// TIA Portal V15.1 export
// export: Created 2024-05-17T05:38:52.6374958Z, ExportSetting WithDefaults, DisplayName Totally Integrated Automation Portal, DisplayVersion V15.1 Update 5, DisplayName TIA Portal Openness, DisplayVersion V15.1 Update 5, DisplayName SINAMICS Startdrive Advanced, DisplayVersion V15.1, DisplayName G130, G150, S120, S150, SINAMICS MV, S210, DisplayVersion V15.1, DisplayName G110M, G120, G120C, G120D, G120P, DisplayVersion V15.1, DisplayName STEP 7 Professional, DisplayVersion V15.1 Update 5, DisplayName STEP 7 Safety, DisplayVersion V15.1, DisplayName WinCC Professional, DisplayVersion V15.1 Update 5, DisplayName SIMATIC Visualization Architect, DisplayVersion V15.1
FUNCTION_BLOCK "LGBTrfOutRel"   // FB6701, FBD
TITLE = LGBTrfOutRel
{ S7_Optimized_Access := 'TRUE' }
VERSION : 0.1
// =============================================================================
// The ReleaseTrfOut function is a FB to be used in transport functions 
// block (as roller, cross-section, …) to release an OUT transfer at an earlier
// stage to gain cycletime in automatic Mode or in manual Mode.
// stored: AutoNumber false, IsIECCheckEnabled false, IsRetainMemResEnabled false, MemoryReserve 100, SetENOAutomatically False, UDAEnableTagReadback false
   VAR_INPUT
      I_TrfOutPrev_TM { ExternalAccessible := 'False'; ExternalVisible := 'False'; ExternalWritable := 'False'} : Bool;   // Transfer communication for outfeed from previous conveyor
      I_TrfOutPrev_RdyDlv { ExternalAccessible := 'False'; ExternalVisible := 'False'; ExternalWritable := 'False'} : Bool;   // Transfer communication for outfeed from previous conveyor
      I_TrfInNext_Arrived { ExternalAccessible := 'False'; ExternalVisible := 'False'; ExternalWritable := 'False'} : Bool;   // Transfer communication for infeed on next conveyor
      I_TrfInNext_RdyRcv { ExternalAccessible := 'False'; ExternalVisible := 'False'; ExternalWritable := 'False'} : Bool;   // Transfer communication for infeed on next conveyor
      I_ReleaseDet { ExternalAccessible := 'False'; ExternalVisible := 'False'; ExternalWritable := 'False'} : Bool;   // Detection to release the outfeed transfer of the previous conveyor
      I_SafetyOk { ExternalAccessible := 'False'; ExternalVisible := 'False'; ExternalWritable := 'False'} : Bool;   // Safety Ok
   END_VAR
   VAR_OUTPUT
      O_TrfOutPrev_Arrived { ExternalAccessible := 'False'; ExternalVisible := 'False'; ExternalWritable := 'False'} : Bool;   // Transfer communication for outfeed from previous conveyor
      O_TrfOutPrev_RdyRcv { ExternalAccessible := 'False'; ExternalVisible := 'False'; ExternalWritable := 'False'} : Bool;   // Transfer communication for outfeed from previous conveyor
      O_TrfInNext_TrfOutCmd { ExternalAccessible := 'False'; ExternalVisible := 'False'; ExternalWritable := 'False'} : Bool;   // Command request after interlock / Command Request after Interlock / Transfer communication for infeed on next conveyor
      O_TrfInNext_TM { ExternalAccessible := 'False'; ExternalVisible := 'False'; ExternalWritable := 'False'} : Bool;   // Transfer communication for infeed on next conveyor
      O_TrfInNext_RdyDlv { ExternalAccessible := 'False'; ExternalVisible := 'False'; ExternalWritable := 'False'} : Bool;   // Transfer communication for infeed on next conveyor
      O_OvertimeAlarm { ExternalAccessible := 'False'; ExternalVisible := 'False'; ExternalWritable := 'False'} : Bool;   // Overtime alarm (0=no alarm / 1=Alarm) / Overtime Alarm
      O_ConfigCalibrationAlm { ExternalAccessible := 'False'; ExternalVisible := 'False'; ExternalWritable := 'False'} : Bool;   // Config/Calibration Alarm
      O_CalibrationWarn { ExternalAccessible := 'False'; ExternalVisible := 'False'; ExternalWritable := 'False'} : Bool;   // Warning Calibration
      O_AlarmABCondition { ExternalAccessible := 'False'; ExternalVisible := 'False'; ExternalWritable := 'False'} : Bool;   // Alarm AB condition / Alarm AB Condition
   END_VAR
   VAR_IN_OUT
      IO_Modes : "Modes";   // Modes
      H_HMI : "H_HMI";   // Animation
      H_TrfOut : "H_TrfOut";   // Animation
      C_TrfMaxTime { ExternalAccessible := 'False'; ExternalVisible := 'False'; ExternalWritable := 'False'} : DInt := 8000;   // Time Delay-On Overtime alarm (millisec) / Time Delay-On Overtime Alarm (millisec)
      C_TrfMaxTimeAfterOvertime { ExternalAccessible := 'False'; ExternalVisible := 'False'; ExternalWritable := 'False'} : DInt := 0;   // Time Delay-On after reset/start after Overtime Alarm (millisec)
      C_EnableTimeoutAlarm { ExternalAccessible := 'False'; ExternalVisible := 'False'; ExternalWritable := 'False'} : Bool;   // Enable Timeout Alarm
   END_VAR
   VAR RETAIN
      Release { ExternalAccessible := 'False'; ExternalVisible := 'False'; ExternalWritable := 'False'} : Bool;   // Memory of release detection negative edge
   END_VAR
   VAR
      Edge { ExternalAccessible := 'False'; ExternalVisible := 'False'; ExternalWritable := 'False'} : Array[0..3] of Bool;   // Edges
      AlarmA { ExternalAccessible := 'False'; ExternalVisible := 'False'; ExternalWritable := 'False'} : Bool;   // Summation Alarm A of roller. / Alarm A
      AlarmB { ExternalAccessible := 'False'; ExternalVisible := 'False'; ExternalWritable := 'False'} : Bool;   // Summation Alarm B of roller. / Alarm B
      AlarmC { ExternalAccessible := 'False'; ExternalVisible := 'False'; ExternalWritable := 'False'} : Bool;   // Summation Alarm C of roller. / Alarm C
      AlarmD { ExternalAccessible := 'False'; ExternalVisible := 'False'; ExternalWritable := 'False'} : Bool;   // Summation Alarm D of roller. / Alarm D
      AlarmABCondition { ExternalAccessible := 'False'; ExternalVisible := 'False'; ExternalWritable := 'False'} : Bool;   // Resetable alarm / Alarm AB Condition
   END_VAR
   VAR RETAIN
      OvertimeAlarm { ExternalAccessible := 'False'; ExternalVisible := 'False'; ExternalWritable := 'False'} : Bool;   // MEM Overtime alarm / MEM Overtime Alarm
      OvertimeAlarmAlmCond { ExternalAccessible := 'False'; ExternalVisible := 'False'; ExternalWritable := 'False'} : Bool;   // MEM Overtime alarm / MEM Overtime Alarm / Overtime Alarm
      TimerOvertimeAlarm { ExternalAccessible := 'False'; ExternalVisible := 'False'; ExternalWritable := 'False'} : Bool;   // MEM Overtime alarm / MEM Overtime Alarm / Overtime Alarm
   END_VAR
   VAR
      TimerOvertimAlarm { ExternalAccessible := 'False'; ExternalVisible := 'False'; ExternalWritable := 'False'} : "LTimer";   // FB
      TrfMaxTime { ExternalAccessible := 'False'; ExternalVisible := 'False'; ExternalWritable := 'False'} : DInt;   // Maximum Transfer Time
      ConfigCalibrationAlm { ExternalAccessible := 'False'; ExternalVisible := 'False'; ExternalWritable := 'False'} : Bool;   // Config/Calibration Alarm
      CalibrationWarn { ExternalAccessible := 'False'; ExternalVisible := 'False'; ExternalWritable := 'False'} : Bool;   // Warning Calibration
   END_VAR
   VAR RETAIN
      OvtTrfMaxTime { ExternalAccessible := 'False'; ExternalVisible := 'False'; ExternalWritable := 'False'} : DInt;   // Alarm Value
      OvtTrfMaxTimeAfterOvertime { ExternalAccessible := 'False'; ExternalVisible := 'False'; ExternalWritable := 'False'} : DInt;   // Alarm Value
      CalibratedTransfer { ExternalAccessible := 'False'; ExternalVisible := 'False'; ExternalWritable := 'False'} : Bool;
   END_VAR
   VAR
      AlarmTimeWithConfig { ExternalAccessible := 'False'; ExternalVisible := 'False'; ExternalWritable := 'False'} : Bool;
      AlarmTimeWithCalibration { ExternalAccessible := 'False'; ExternalVisible := 'False'; ExternalWritable := 'False'} : Bool;
   END_VAR
   VAR_TEMP
      H_CalibrateTransfer : Bool;   // HMI Function
      TempReal : Real;
   END_VAR
   VAR_TEMP   // added for the SCL form of the ladder/FBD networks
      _w1 : Bool;
      _w2 : Bool;
      _w3 : Bool;
      _w4 : Bool;
   END_VAR
BEGIN

REGION Network 1: **** 1 - Inputs **** HMI Commands
   // Extract the Commands from HMIRobCmd / Extract the Commands from HMI
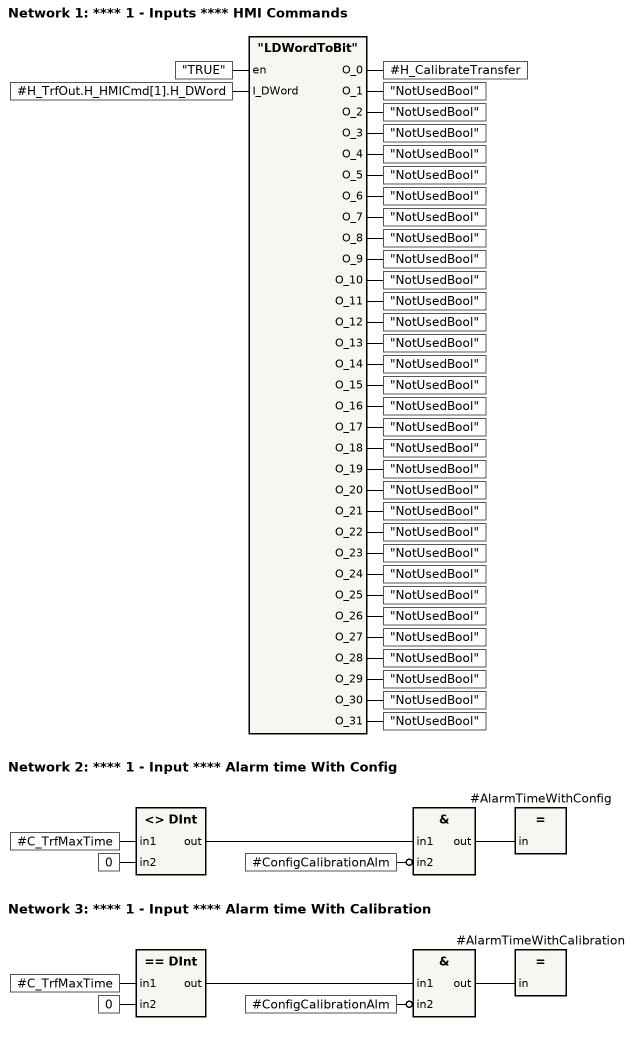
   IF "TRUE" THEN
       "LDWordToBit"(I_DWord := #H_TrfOut.H_HMICmd[1].H_DWord,
                     O_0 => #H_CalibrateTransfer,
                     O_1 => "NotUsedBool",
                     O_2 => "NotUsedBool",
                     O_3 => "NotUsedBool",
                     O_4 => "NotUsedBool",
                     O_5 => "NotUsedBool",
                     O_6 => "NotUsedBool",
                     O_7 => "NotUsedBool",
                     O_8 => "NotUsedBool",
                     O_9 => "NotUsedBool",
                     O_10 => "NotUsedBool",
                     O_11 => "NotUsedBool",
                     O_12 => "NotUsedBool",
                     O_13 => "NotUsedBool",
                     O_14 => "NotUsedBool",
                     O_15 => "NotUsedBool",
                     O_16 => "NotUsedBool",
                     O_17 => "NotUsedBool",
                     O_18 => "NotUsedBool",
                     O_19 => "NotUsedBool",
                     O_20 => "NotUsedBool",
                     O_21 => "NotUsedBool",
                     O_22 => "NotUsedBool",
                     O_23 => "NotUsedBool",
                     O_24 => "NotUsedBool",
                     O_25 => "NotUsedBool",
                     O_26 => "NotUsedBool",
                     O_27 => "NotUsedBool",
                     O_28 => "NotUsedBool",
                     O_29 => "NotUsedBool",
                     O_30 => "NotUsedBool",
                     O_31 => "NotUsedBool");
   END_IF;
END_REGION

REGION Network 2: **** 1 - Input **** Alarm time With Config
   #AlarmTimeWithConfig := (#C_TrfMaxTime <> 0) AND NOT #ConfigCalibrationAlm;
END_REGION

REGION Network 3: **** 1 - Input **** Alarm time With Calibration
   #AlarmTimeWithCalibration := (#C_TrfMaxTime = 0) AND NOT #ConfigCalibrationAlm;
END_REGION

REGION Network 4: Calibrated Set / **** 1 - Input **** Ovt Values / **** 1 - Inputs **** Ovt Values
   // Ovt Values
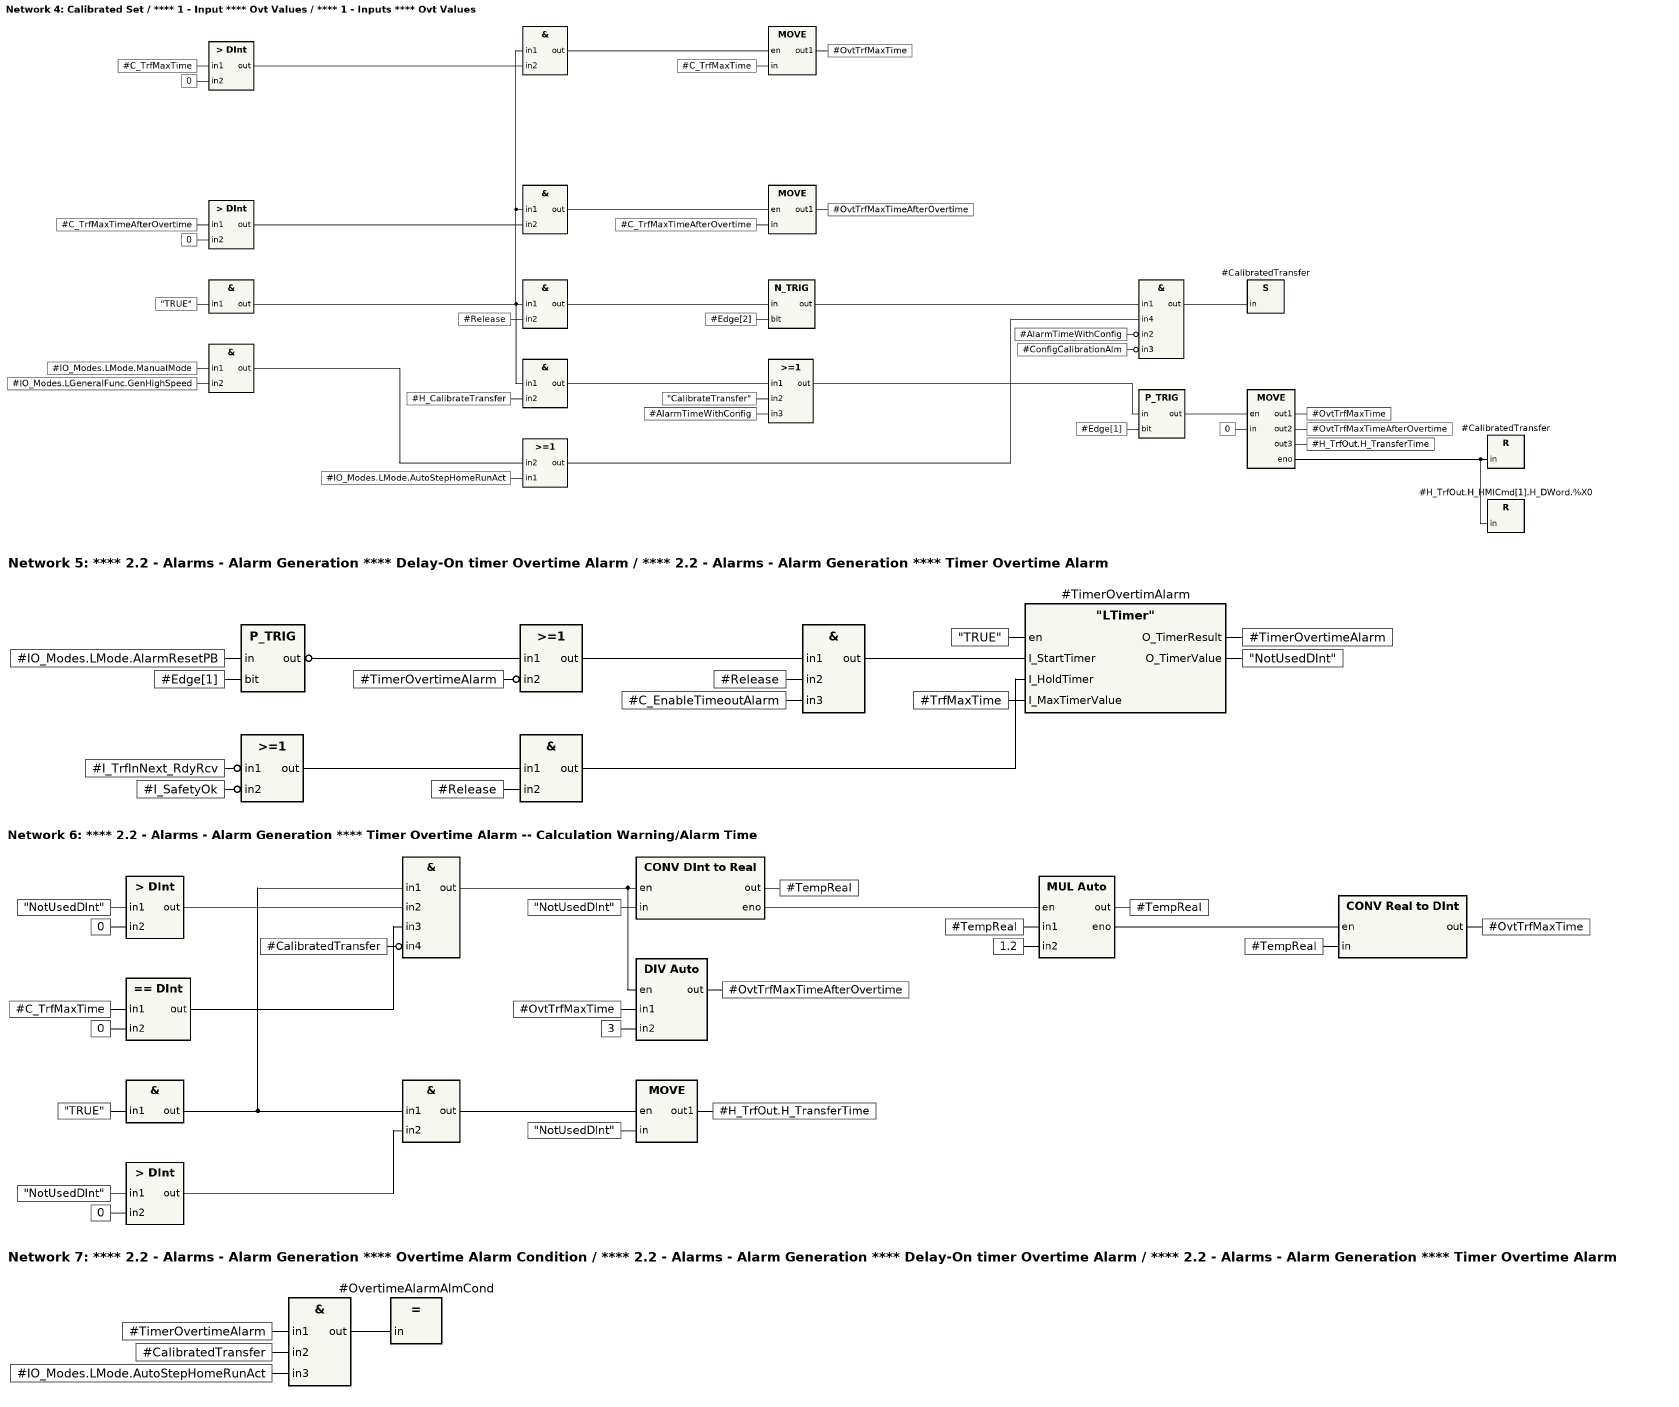
   // ENO of a box is taken as its EN; it also drops when the box reports an error
   IF "TRUE" AND (#C_TrfMaxTime > 0) THEN #OvtTrfMaxTime := #C_TrfMaxTime; END_IF;
   IF "TRUE" AND (#C_TrfMaxTimeAfterOvertime > 0) THEN
       #OvtTrfMaxTimeAfterOvertime := #C_TrfMaxTimeAfterOvertime;
   END_IF;
   #_w1 := "TRUE" AND #Release;
   #_w2 := NOT #_w1 AND #Edge[2];   // falling edge
   #Edge[2] := #_w1;
   IF #_w2 AND ((#IO_Modes.LMode.ManualMode AND #IO_Modes.LGeneralFunc.GenHighSpeed) OR #IO_Modes.LMode.AutoStepHomeRunAct) AND NOT #AlarmTimeWithConfig AND NOT #ConfigCalibrationAlm THEN
       #CalibratedTransfer := TRUE;
   END_IF;
   #_w3 := ("TRUE" AND #H_CalibrateTransfer) OR "CalibrateTransfer" OR #AlarmTimeWithConfig;
   #_w4 := #_w3 AND NOT #Edge[1];   // rising edge
   #Edge[1] := #_w3;
   IF #_w4 THEN
       #OvtTrfMaxTime := 0;
       #OvtTrfMaxTimeAfterOvertime := 0;
       #H_TrfOut.H_TransferTime := 0;
       #CalibratedTransfer := FALSE;
       #H_TrfOut.H_HMICmd[1].H_DWord.%X0 := FALSE;
   END_IF;
END_REGION

REGION Network 5: **** 2.2 - Alarms - Alarm Generation **** Delay-On timer Overtime Alarm / **** 2.2 - Alarms - Alarm Generation **** Timer Overtime Alarm
   // Delay-On timer Overtime Alarm
   #_w1 := #IO_Modes.LMode.AlarmResetPB AND NOT #Edge[1];   // rising edge
   #Edge[1] := #IO_Modes.LMode.AlarmResetPB;
   IF "TRUE" THEN
       #TimerOvertimAlarm(I_StartTimer := (NOT #_w1 OR NOT #TimerOvertimeAlarm) AND #Release AND #C_EnableTimeoutAlarm,   // "LTimer"
                          I_HoldTimer := (NOT #I_TrfInNext_RdyRcv OR NOT #I_SafetyOk) AND #Release,
                          I_MaxTimerValue := #TrfMaxTime,
                          O_TimerResult => #TimerOvertimeAlarm,
                          O_TimerValue => "NotUsedDInt");
   END_IF;
END_REGION

REGION Network 6: **** 2.2 - Alarms - Alarm Generation **** Timer Overtime Alarm -- Calculation Warning/Alarm Time
   IF "TRUE" AND ("NotUsedDInt" > 0) AND (#C_TrfMaxTime = 0) AND NOT #CalibratedTransfer THEN
       #TempReal := DINT_TO_REAL("NotUsedDInt");
       #TempReal := #TempReal * 1.2;
       #OvtTrfMaxTime := REAL_TO_DINT(#TempReal);
       #OvtTrfMaxTimeAfterOvertime := #OvtTrfMaxTime / 3;
   END_IF;
   IF "TRUE" AND ("NotUsedDInt" > 0) THEN #H_TrfOut.H_TransferTime := "NotUsedDInt"; END_IF;
END_REGION

REGION Network 7: **** 2.2 - Alarms - Alarm Generation **** Overtime Alarm Condition / **** 2.2 - Alarms - Alarm Generation **** Delay-On timer Overtime Alarm / **** 2.2 - Alarms - Alarm Generation **** Timer Overtime Alarm
   // Delay-On timer Overtime Alarm
   #OvertimeAlarmAlmCond := #TimerOvertimeAlarm AND #CalibratedTransfer AND #IO_Modes.LMode.AutoStepHomeRunAct;
END_REGION

REGION Network 8: **** 2.2 - Alarms - Alarm Generation **** OverTime Alarm / **** 2.2 - Alarms - Alarm Generation **** Overrtime Alarm
   // Overrtime Alarm
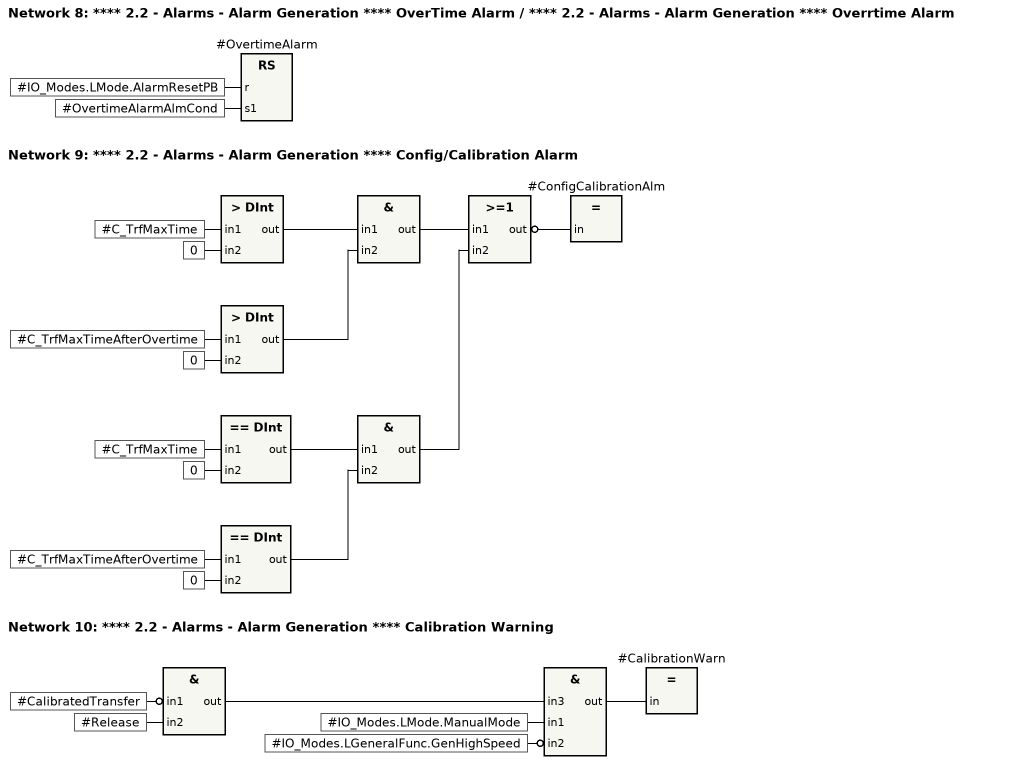
   IF #IO_Modes.LMode.AlarmResetPB THEN
       #OvertimeAlarm := FALSE;   // RS flip-flop
   END_IF;
   IF #OvertimeAlarmAlmCond THEN #OvertimeAlarm := TRUE; END_IF;
END_REGION

REGION Network 9: **** 2.2 - Alarms - Alarm Generation **** Config/Calibration Alarm
   #ConfigCalibrationAlm := NOT (((#C_TrfMaxTime > 0) AND (#C_TrfMaxTimeAfterOvertime > 0)) OR ((#C_TrfMaxTime = 0) AND (#C_TrfMaxTimeAfterOvertime = 0)));
END_REGION

REGION Network 10: **** 2.2 - Alarms - Alarm Generation **** Calibration Warning
   #CalibrationWarn := NOT #CalibratedTransfer AND #Release AND #IO_Modes.LMode.ManualMode AND NOT #IO_Modes.LGeneralFunc.GenHighSpeed;
END_REGION

REGION Network 11: **** 4.6 - Machine Status - Indication **** Icon Animation
   // Icon Animation
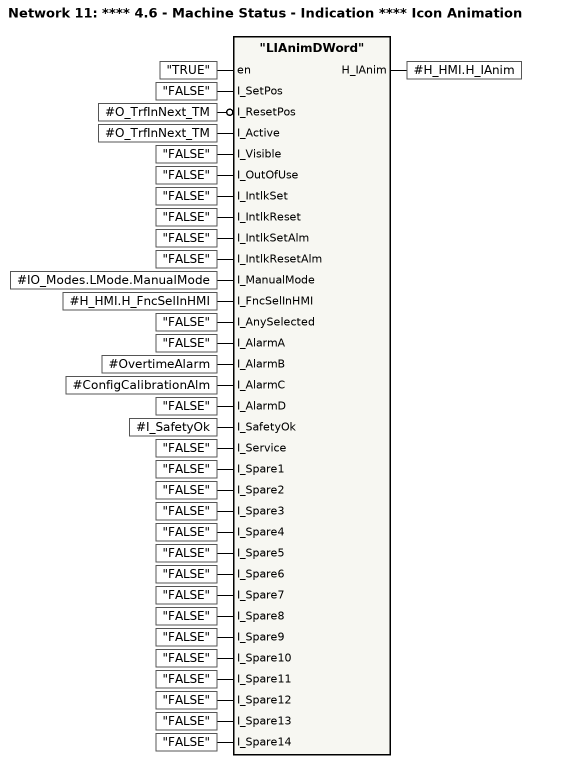
   IF "TRUE" THEN
       "LIAnimDWord"(I_SetPos := "FALSE",
                     I_ResetPos := NOT #O_TrfInNext_TM,
                     I_Active := #O_TrfInNext_TM,
                     I_Visible := "FALSE",
                     I_OutOfUse := "FALSE",
                     I_IntlkSet := "FALSE",
                     I_IntlkReset := "FALSE",
                     I_IntlkSetAlm := "FALSE",
                     I_IntlkResetAlm := "FALSE",
                     I_ManualMode := #IO_Modes.LMode.ManualMode,
                     I_FncSelInHMI := #H_HMI.H_FncSelInHMI,
                     I_AnySelected := "FALSE",
                     I_AlarmA := "FALSE",
                     I_AlarmB := #OvertimeAlarm,
                     I_AlarmC := #ConfigCalibrationAlm,
                     I_AlarmD := "FALSE",
                     I_SafetyOk := #I_SafetyOk,
                     I_Service := "FALSE",
                     I_Spare1 := "FALSE",
                     I_Spare2 := "FALSE",
                     I_Spare3 := "FALSE",
                     I_Spare4 := "FALSE",
                     I_Spare5 := "FALSE",
                     I_Spare6 := "FALSE",
                     I_Spare7 := "FALSE",
                     I_Spare8 := "FALSE",
                     I_Spare9 := "FALSE",
                     I_Spare10 := "FALSE",
                     I_Spare11 := "FALSE",
                     I_Spare12 := "FALSE",
                     I_Spare13 := "FALSE",
                     I_Spare14 := "FALSE",
                     H_IAnim => #H_HMI.H_IAnim);
   END_IF;
END_REGION

REGION Network 12: **** 4.6 - Machine Status - Indication **** Animation
   // Animation
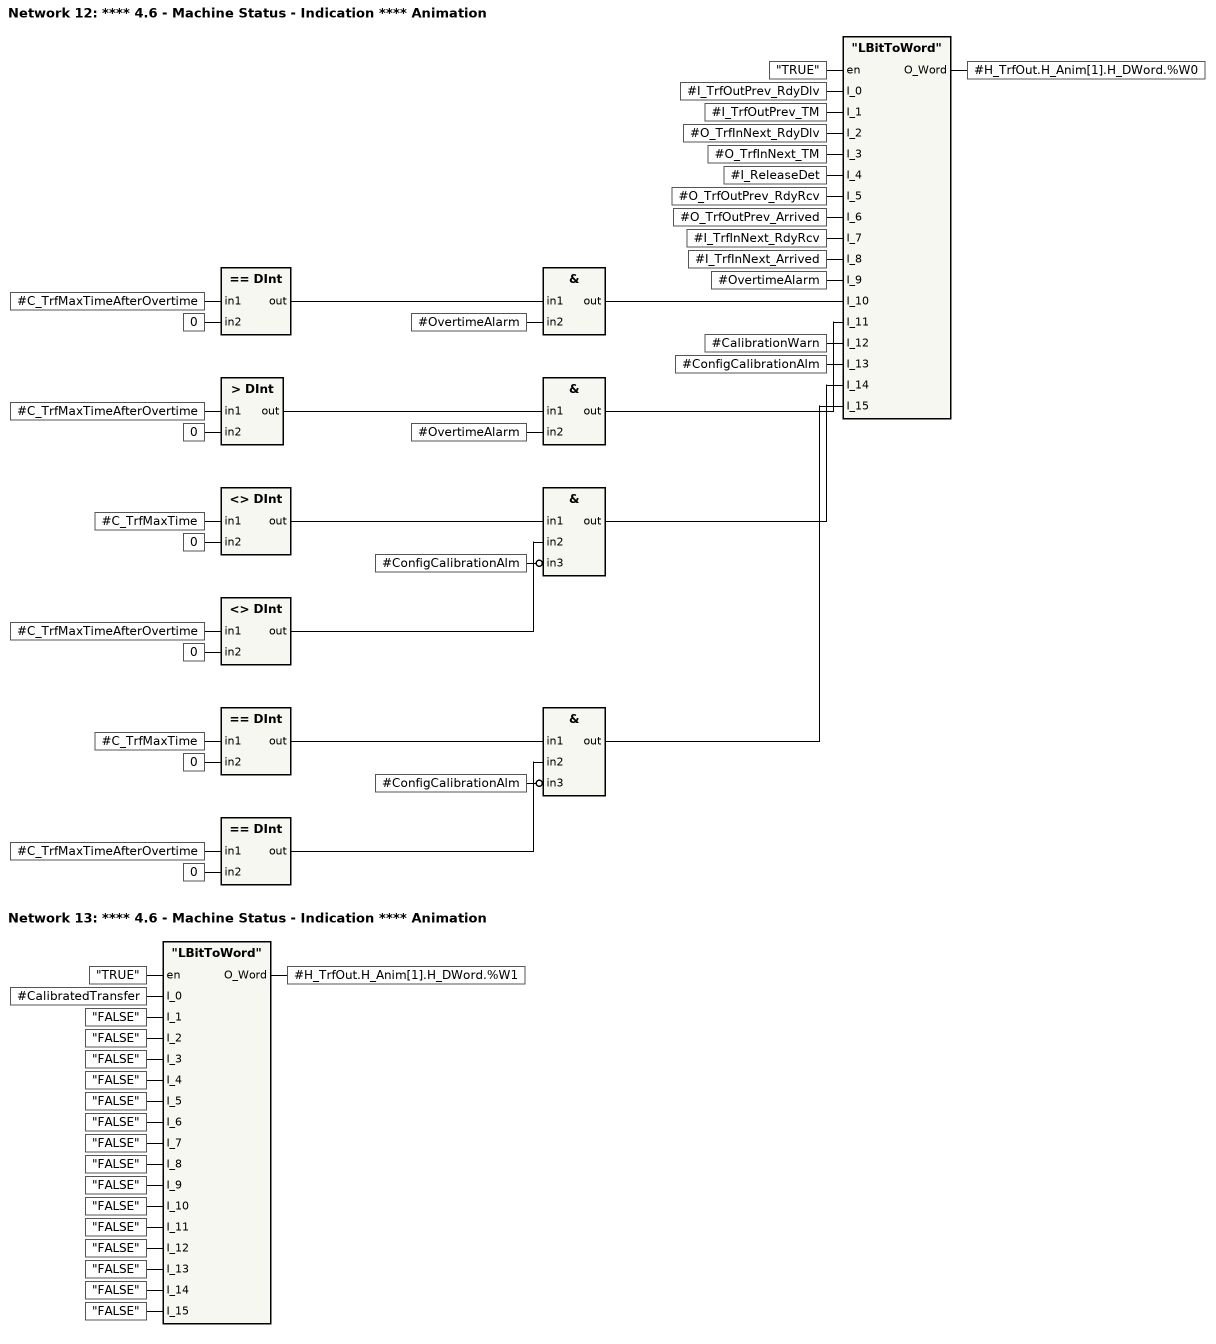
   IF "TRUE" THEN
       "LBitToWord"(I_0 := #I_TrfOutPrev_RdyDlv,
                    I_1 := #I_TrfOutPrev_TM,
                    I_2 := #O_TrfInNext_RdyDlv,
                    I_3 := #O_TrfInNext_TM,
                    I_4 := #I_ReleaseDet,
                    I_5 := #O_TrfOutPrev_RdyRcv,
                    I_6 := #O_TrfOutPrev_Arrived,
                    I_7 := #I_TrfInNext_RdyRcv,
                    I_8 := #I_TrfInNext_Arrived,
                    I_9 := #OvertimeAlarm,
                    I_10 := (#C_TrfMaxTimeAfterOvertime = 0) AND #OvertimeAlarm,
                    I_11 := (#C_TrfMaxTimeAfterOvertime > 0) AND #OvertimeAlarm,
                    I_12 := #CalibrationWarn,
                    I_13 := #ConfigCalibrationAlm,
                    I_14 := (#C_TrfMaxTime <> 0) AND (#C_TrfMaxTimeAfterOvertime <> 0) AND NOT #ConfigCalibrationAlm,
                    I_15 := (#C_TrfMaxTime = 0) AND (#C_TrfMaxTimeAfterOvertime = 0) AND NOT #ConfigCalibrationAlm,
                    O_Word => #H_TrfOut.H_Anim[1].H_DWord.%W0);
   END_IF;
END_REGION

REGION Network 13: **** 4.6 - Machine Status - Indication **** Animation
   // Animation
   IF "TRUE" THEN
       "LBitToWord"(I_0 := #CalibratedTransfer,
                    I_1 := "FALSE",
                    I_2 := "FALSE",
                    I_3 := "FALSE",
                    I_4 := "FALSE",
                    I_5 := "FALSE",
                    I_6 := "FALSE",
                    I_7 := "FALSE",
                    I_8 := "FALSE",
                    I_9 := "FALSE",
                    I_10 := "FALSE",
                    I_11 := "FALSE",
                    I_12 := "FALSE",
                    I_13 := "FALSE",
                    I_14 := "FALSE",
                    I_15 := "FALSE",
                    O_Word => #H_TrfOut.H_Anim[1].H_DWord.%W1);
   END_IF;
END_REGION

REGION Network 14: **** 4.6 - Machine Status - Indication **** Animation
   // Animation
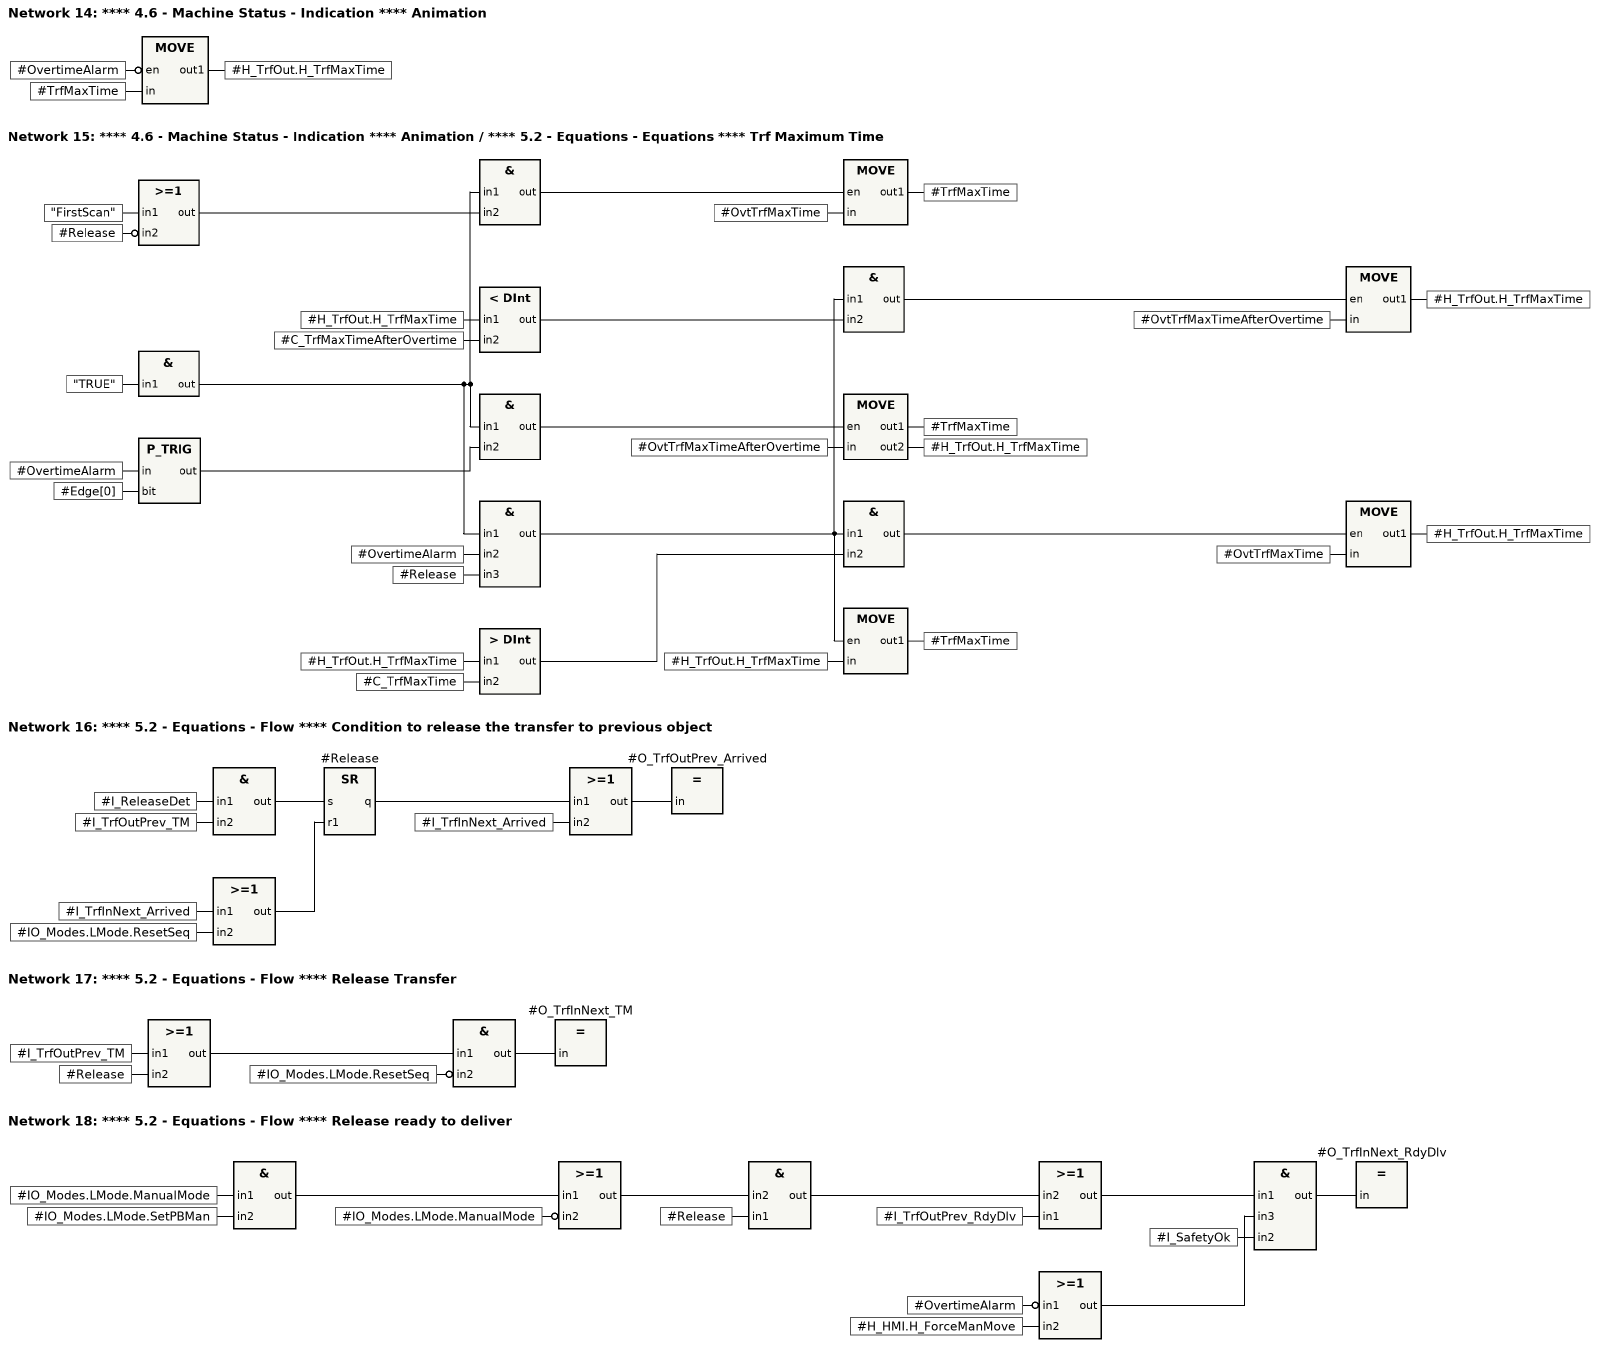
   IF NOT #OvertimeAlarm THEN #H_TrfOut.H_TrfMaxTime := #TrfMaxTime; END_IF;
END_REGION

REGION Network 15: **** 4.6 - Machine Status - Indication **** Animation / **** 5.2 - Equations - Equations **** Trf Maximum Time
   // Animation / Trf Maximum Time
   IF "TRUE" AND ("FirstScan" OR NOT #Release) THEN #TrfMaxTime := #OvtTrfMaxTime; END_IF;
   #_w1 := #OvertimeAlarm AND NOT #Edge[0];   // rising edge
   #Edge[0] := #OvertimeAlarm;
   IF "TRUE" AND #_w1 THEN
       #TrfMaxTime := #OvtTrfMaxTimeAfterOvertime;
       #H_TrfOut.H_TrfMaxTime := #OvtTrfMaxTimeAfterOvertime;
   END_IF;
   #_w2 := "TRUE" AND #OvertimeAlarm AND #Release;
   IF #_w2 AND (#H_TrfOut.H_TrfMaxTime < #C_TrfMaxTimeAfterOvertime) THEN
       #H_TrfOut.H_TrfMaxTime := #OvtTrfMaxTimeAfterOvertime;
   END_IF;
   IF #_w2 AND (#H_TrfOut.H_TrfMaxTime > #C_TrfMaxTime) THEN
       #H_TrfOut.H_TrfMaxTime := #OvtTrfMaxTime;
   END_IF;
   IF #_w2 THEN #TrfMaxTime := #H_TrfOut.H_TrfMaxTime; END_IF;
END_REGION

REGION Network 16: **** 5.2 - Equations - Flow **** Condition to release the transfer to previous object
   // Condition to release the transfer to previous object
   IF #I_ReleaseDet AND #I_TrfOutPrev_TM THEN
       #Release := TRUE;   // SR flip-flop
   END_IF;
   IF #I_TrfInNext_Arrived OR #IO_Modes.LMode.ResetSeq THEN #Release := FALSE; END_IF;
   #O_TrfOutPrev_Arrived := #Release OR #I_TrfInNext_Arrived;
END_REGION

REGION Network 17: **** 5.2 - Equations - Flow **** Release Transfer
   // The signal Transfer of next object starts with the signal from previous and continues until the arrived signal is formed
   #O_TrfInNext_TM := (#I_TrfOutPrev_TM OR #Release) AND NOT #IO_Modes.LMode.ResetSeq;
END_REGION

REGION Network 18: **** 5.2 - Equations - Flow **** Release ready to deliver
   // The signal Ready deliver of next object starts with the signal from previous roller and continues until the arrived signal is formed
   #O_TrfInNext_RdyDlv := ((((#IO_Modes.LMode.ManualMode AND #IO_Modes.LMode.SetPBMan) OR NOT #IO_Modes.LMode.ManualMode) AND #Release) OR #I_TrfOutPrev_RdyDlv) AND (NOT #OvertimeAlarm OR #H_HMI.H_ForceManMove) AND #I_SafetyOk;
END_REGION

REGION Network 19: **** 5.2 - Equations - Flow **** Connect TrfIn Ready to receive to TrfOut Ready To Receive
   // Connnect TrfInNextPrev to TrfOutPrev
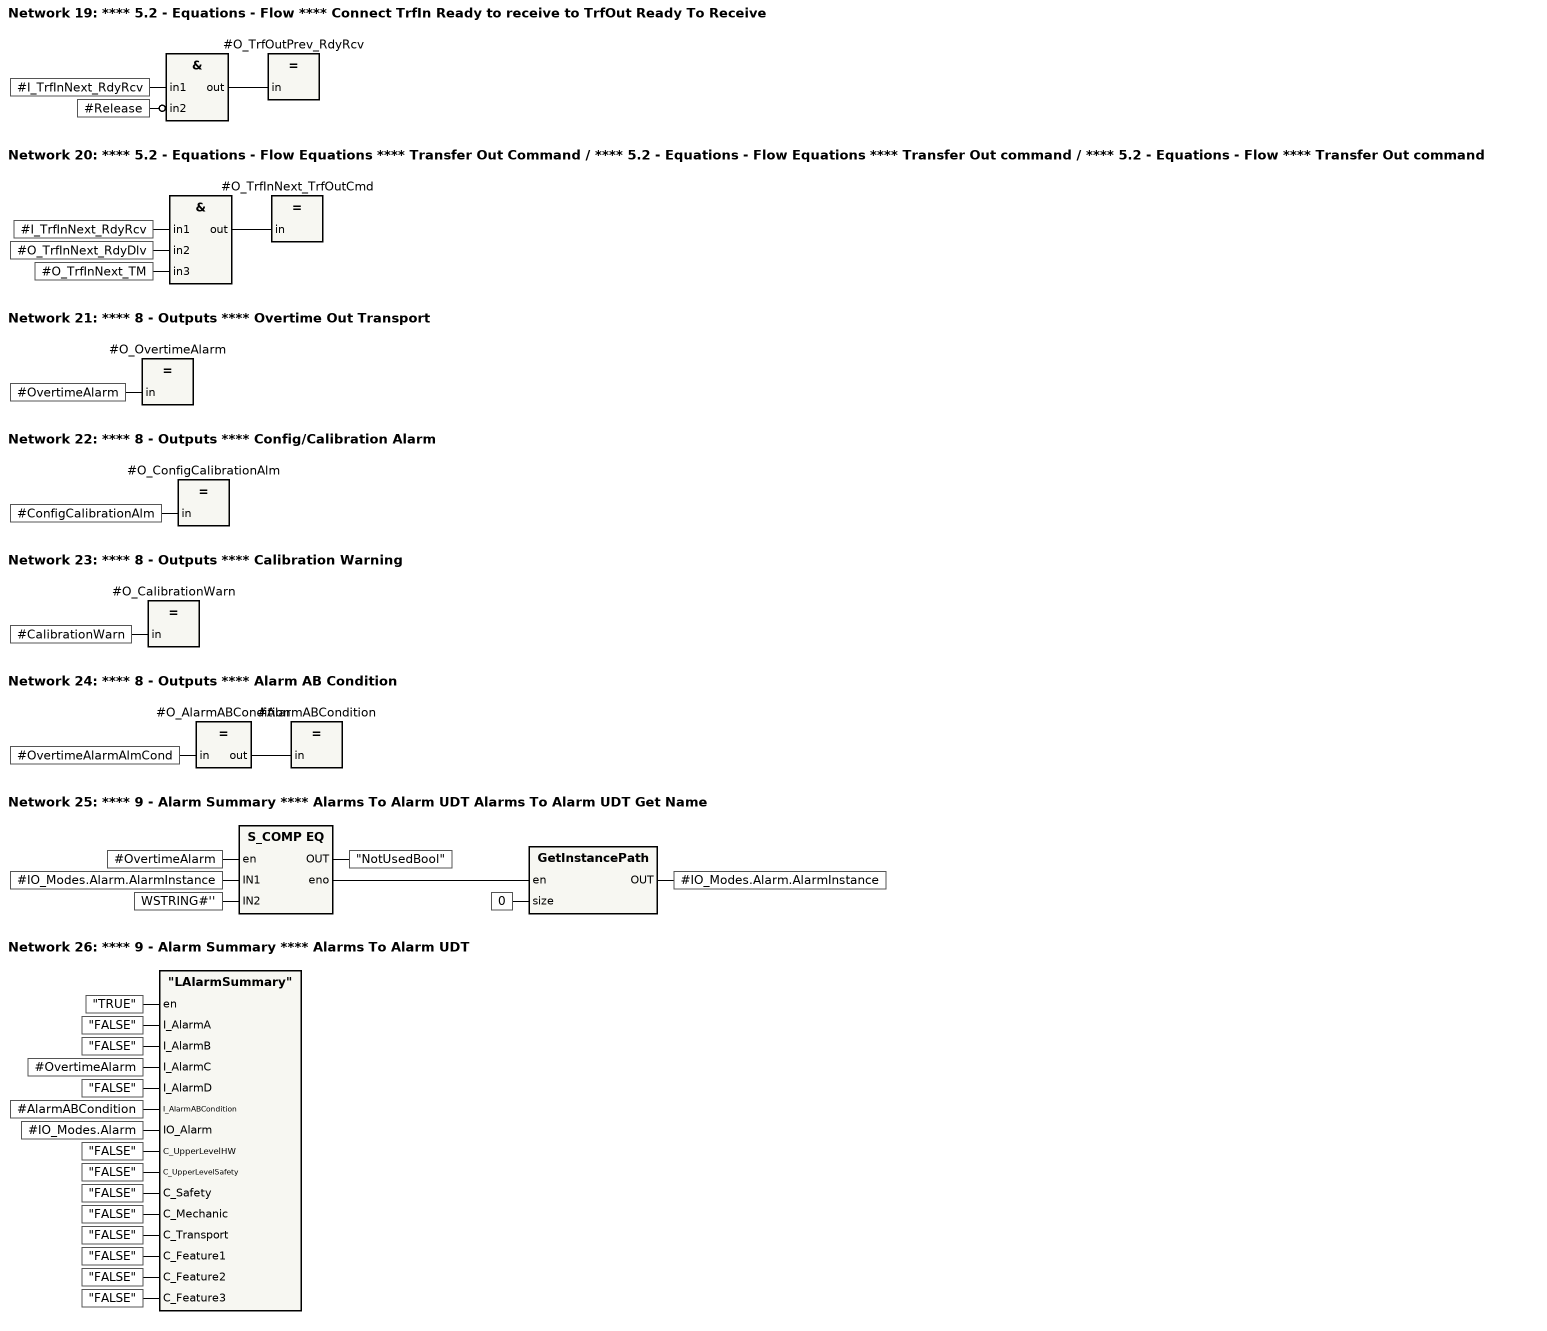
   #O_TrfOutPrev_RdyRcv := #I_TrfInNext_RdyRcv AND NOT #Release;
END_REGION

REGION Network 20: **** 5.2 - Equations - Flow Equations **** Transfer Out Command / **** 5.2 - Equations - Flow Equations **** Transfer Out command / **** 5.2 - Equations - Flow **** Transfer Out command
   // Transfer Out Command / Transfer Out command
   #O_TrfInNext_TrfOutCmd := #I_TrfInNext_RdyRcv AND #O_TrfInNext_RdyDlv AND #O_TrfInNext_TM;
END_REGION

REGION Network 21: **** 8 - Outputs **** Overtime Out Transport
   // Overtime Out Transport
   #O_OvertimeAlarm := #OvertimeAlarm;
END_REGION

REGION Network 22: **** 8 - Outputs **** Config/Calibration Alarm
   #O_ConfigCalibrationAlm := #ConfigCalibrationAlm;
END_REGION

REGION Network 23: **** 8 - Outputs **** Calibration Warning
   #O_CalibrationWarn := #CalibrationWarn;
END_REGION

REGION Network 24: **** 8 - Outputs **** Alarm AB Condition
   // Alarm AB Condition
   #O_AlarmABCondition := #OvertimeAlarmAlmCond;
   #AlarmABCondition := #OvertimeAlarmAlmCond;
END_REGION

REGION Network 25: **** 9 - Alarm Summary **** Alarms To Alarm UDT Alarms To Alarm UDT Get Name
   // Alarm / Alarm D
   S_COMP(EN := #OvertimeAlarm,
          IN1 := #IO_Modes.Alarm.AlarmInstance,
          IN2 := WSTRING#'',
          OUT => "NotUsedBool",
          ENO => #_w1);
   IF #_w1 THEN GetInstancePath(size := 0, OUT => #IO_Modes.Alarm.AlarmInstance); END_IF;
END_REGION

REGION Network 26: **** 9 - Alarm Summary **** Alarms To Alarm UDT
   // Alarm / Alarm D
   IF "TRUE" THEN
       "LAlarmSummary"(I_AlarmA := "FALSE",
                       I_AlarmB := "FALSE",
                       I_AlarmC := #OvertimeAlarm,
                       I_AlarmD := "FALSE",
                       I_AlarmABCondition := #AlarmABCondition,
                       IO_Alarm := #IO_Modes.Alarm,
                       C_UpperLevelHW := "FALSE",
                       C_UpperLevelSafety := "FALSE",
                       C_Safety := "FALSE",
                       C_Mechanic := "FALSE",
                       C_Transport := "FALSE",
                       C_Feature1 := "FALSE",
                       C_Feature2 := "FALSE",
                       C_Feature3 := "FALSE");
   END_IF;
END_REGION
END_FUNCTION_BLOCK
